{attribute 'hide_all_locals'}
FUNCTION_BLOCK FB_3_COMM_AXIS_BECKHOFF EXTENDS FB_1_COMM
VAR_INPUT
  StopVelocityTolerance : LREAL := 0.000001;
END_VAR
VAR_IN_OUT
    Axis : AXIS_REF;
END_VAR
VAR_OUTPUT
  Powered : BOOL;
  Homed : BOOL;
  ActualPosition : LREAL;
  ActualVelocity : LREAL;
END_VAR
VAR
    _fbPower : MC_Power;
    _fbMoveAbsolute : MC_MoveAbsolute;
    _fbMoveRelative : MC_MoveRelative;
    _fbHome : MC_Home;
    _fbStop : MC_Stop;
    _fbReset : MC_Reset;

    _powerRequest : BOOL;
    _moveAbsExecute : BOOL;
    _moveRelExecute : BOOL;
    _homeExecute : BOOL;
    _stopExecute : BOOL;
    _resetExecute : BOOL;
    _commandAccepted : BOOL;
END_VAR

// ------ CALL CYCLIC -----------------
CYCLIC_COMM();



// ------ WRITE HMI -------------------
		// NO HMI STRUCT

// ------ READ FROM HMI ---------------
		// NO HMI STRUCT
	


// ------ WRITE PROPS/METHODS ---------
Connected := RequestConnection;
Operational := RequestConnection;

CanAcceptCommand := NOT _fbStop.Busy AND NOT _stopExecute AND NOT _resetExecute;


// ----- CALL POUS AND ERROR SURVEILLANCE ----------

_fbPower(Axis := Axis, Enable := _powerRequest, Enable_Positive := _powerRequest, Enable_Negative := _powerRequest);
_fbMoveAbsolute(Axis := Axis, Execute := _moveAbsExecute);
_fbMoveRelative(Axis := Axis, Execute := _moveRelExecute);
_fbHome(Axis := Axis, Execute := _homeExecute);
_fbStop(Axis := Axis, Execute := _stopExecute);
_fbReset(Axis := Axis, Execute := _resetExecute);



IF _fbPower.Error THEN Messenger.AddError(eMessageCategories.HardwareFailure, CONCAT(Path, '.Power'), 'MC_Power error'); END_IF
IF _fbMoveAbsolute.Error THEN Messenger.AddError(eMessageCategories.HardwareFailure, CONCAT(Path, '.MoveAbsolute'), 'MC_MoveAbsolute error'); END_IF
IF _fbMoveRelative.Error THEN Messenger.AddError(eMessageCategories.HardwareFailure, CONCAT(Path, '.MoveRelative'), 'MC_MoveRelative error'); END_IF
IF _fbHome.Error THEN Messenger.AddError(eMessageCategories.HardwareFailure, CONCAT(Path, '.Home'), 'MC_Home error'); END_IF
IF _fbStop.Error THEN Messenger.AddError(eMessageCategories.HardwareFailure, CONCAT(Path, '.Stop'), 'MC_Stop error'); END_IF
IF _fbReset.Error THEN Messenger.AddError(eMessageCategories.HardwareFailure, CONCAT(Path, '.Reset'), 'MC_Reset error'); END_IF


// ----- REST --------------------

Powered := _fbPower.Status;
ActualPosition := Axis.NcToPlc.ActPos;
ActualVelocity := Axis.NcToPlc.ActVelo;


IF Busy AND NOT StopPending THEN
  IF Messenger.HasActivError OR NOT Operational THEN
        _moveAbsExecute := FALSE;
        _moveRelExecute := FALSE;
        _homeExecute := FALSE;
        ActiveCommandID := 0;
        CommandState := eProgress.FINALIZED;
        CommandResult :=eResult.ERROR;
        Busy := FALSE;

    ELSIF _fbMoveAbsolute.CommandAborted OR _fbMoveRelative.CommandAborted OR _fbHome.CommandAborted THEN
        _moveAbsExecute := FALSE;
        _moveRelExecute := FALSE;
        _homeExecute := FALSE;
        ActiveCommandID := 0;
        CommandState := eProgress.ABORTED;
        CommandResult :=eResult.FAILURE;
        Busy := FALSE;

    ELSIF _fbMoveAbsolute.Done OR _fbMoveRelative.Done OR _fbHome.Done THEN
        IF _fbHome.Done THEN Homed := TRUE; END_IF
        _moveAbsExecute := FALSE;
        _moveRelExecute := FALSE;
        _homeExecute := FALSE;
        ActiveCommandID := 0;
        CommandState := eProgress.FINALIZED;
        CommandResult :=eResult.SUCCESS;
        Busy := FALSE;

    ELSIF NOT _commandAccepted AND (_fbMoveAbsolute.Busy OR _fbMoveRelative.Busy OR _fbHome.Busy) THEN
        _commandAccepted := TRUE;
        AcceptedCommandID := ActiveCommandID;
        CommandState := eProgress.ACKNOWLEDGE;
        _moveAbsExecute := FALSE;
        _moveRelExecute := FALSE;
        _homeExecute := FALSE;
    ELSIF _commandAccepted AND (_fbMoveAbsolute.Busy OR _fbMoveRelative.Busy OR _fbHome.Busy) THEN
        CommandState := eProgress.RUNNING;
    END_IF
END_IF

IF _fbStop.Done OR _fbStop.CommandAborted OR _fbStop.Error THEN _stopExecute := FALSE; END_IF
IF _fbReset.Done OR _fbReset.Error THEN _resetExecute := FALSE; END_IF

METHOD PROTECTED HasPhysicalStopFailed : BOOL
HasPhysicalStopFailed := _fbStop.Error OR _fbStop.CommandAborted;
END_METHOD

METHOD PROTECTED IsPhysicalStopComplete : BOOL
IsPhysicalStopComplete :=
    _fbStop.Done
    AND (ABS(ActualVelocity) <= StopVelocityTolerance);
END_METHOD

PROPERTY Operational : BOOL
SET
SUPER^.Operational := Operational;
END_SET
END_PROPERTY

METHOD PUBLIC Power : BOOL
VAR_INPUT Enable : BOOL; END_VAR
_powerRequest := Enable;
Power := TRUE;
END_METHOD

METHOD PUBLIC ResetAxis : BOOL
_resetExecute := TRUE;
ResetAxis := TRUE;
END_METHOD

METHOD PUBLIC ResetCommunication : BOOL
_moveAbsExecute := FALSE;
_moveRelExecute := FALSE;
_homeExecute := FALSE;
_stopExecute := FALSE;
AcceptedCommandID := 0;
ActiveCommandID := 0;

CommandState := eProgress.INIT;
CommandResult :=eResult.NONE;
Reconnect();
ResetCommunication := TRUE;
END_METHOD

METHOD PUBLIC SendHome : BOOL
VAR_INPUT CommandID : UINT; END_VAR
SendHome := FALSE;
IF (CommandID = 0) OR NOT CanAcceptCommand THEN RETURN; END_IF
Homed := FALSE;
_homeExecute := TRUE;
_commandAccepted := FALSE;
AcceptedCommandID := 0;
ActiveCommandID := CommandID;
CommandState := eProgress.INIT;
CommandResult :=eResult.NONE;
SendHome := TRUE;
END_METHOD

METHOD PUBLIC SendMoveAbsolute : BOOL
VAR_INPUT
    CommandID : UINT; Position : LREAL; Velocity : LREAL; Acceleration : LREAL; Deceleration : LREAL; Jerk : LREAL;
END_VAR
SendMoveAbsolute := FALSE;
IF (CommandID = 0) OR NOT CanAcceptCommand THEN RETURN; END_IF
_fbMoveAbsolute.Position := Position;
_fbMoveAbsolute.Velocity := Velocity;
_fbMoveAbsolute.Acceleration := Acceleration;
_fbMoveAbsolute.Deceleration := Deceleration;
_fbMoveAbsolute.Jerk := Jerk;
_moveAbsExecute := TRUE;
_commandAccepted := FALSE;
AcceptedCommandID := 0;
ActiveCommandID := CommandID;
CommandState := eProgress.INIT;
CommandResult :=eResult.NONE;
SendMoveAbsolute := TRUE;
END_METHOD

METHOD PUBLIC SendMoveRelative : BOOL
VAR_INPUT
    CommandID : UINT; Distance : LREAL; Velocity : LREAL; Acceleration : LREAL; Deceleration : LREAL; Jerk : LREAL;
END_VAR
SendMoveRelative := FALSE;
IF (CommandID = 0) OR NOT CanAcceptCommand THEN RETURN; END_IF
_fbMoveRelative.Distance := Distance;
_fbMoveRelative.Velocity := Velocity;
_fbMoveRelative.Acceleration := Acceleration;
_fbMoveRelative.Deceleration := Deceleration;
_fbMoveRelative.Jerk := Jerk;
_moveRelExecute := TRUE;
_commandAccepted := FALSE;
AcceptedCommandID := 0;
ActiveCommandID := CommandID;
CommandState := eProgress.INIT;
CommandResult :=eResult.NONE;
SendMoveRelative := TRUE;
END_METHOD

METHOD PROTECTED StartPhysicalStop : BOOL
VAR_INPUT
    Mode : eStopMode;
END_VAR
StartPhysicalStop := FALSE;
IF NOT Connected THEN
    RETURN;
END_IF

_moveAbsExecute := FALSE;
_moveRelExecute := FALSE;
_homeExecute := FALSE;
_stopExecute := TRUE;
StartPhysicalStop := TRUE;
END_METHOD

METHOD PUBLIC StopMotion : BOOL
StopMotion := SUPER^.StopMotion();
END_METHOD

END_FUNCTION_BLOCK

(* stored: Version 1.1.0.1, ProductVersion 3.1.4026.18
   POU FB_3_COMM_AXIS_BECKHOFF: Id {6590ca91-e828-49ed-96d5-a1b6fe08b87c}, SpecialFunc None
   Method HasPhysicalStopFailed: Id {07ba1865-cb6a-4a8c-96a0-eef840195aa0}
   Method IsPhysicalStopComplete: Id {a22113a2-02df-430f-b71d-3b7827035089}
   Property Operational: Id {4e3d4c82-6c3e-4a6a-814a-07ce7bf49eff}
   Set Set: Id {a12a9d16-3a48-4fe1-b1c6-4b5bb26f80c2}
   Method Power: Id {5009c6e1-2c2e-4e9f-8bd0-48ea7245eeb8}
   Method ResetAxis: Id {8993a558-2273-4b75-9edd-81b579dc1f02}
   Method ResetCommunication: Id {d6df4f8c-4fb8-47c4-8972-2548e217db7f}
   Method SendHome: Id {bc5b9968-2431-457c-aab0-516da2c5d033}
   Method SendMoveAbsolute: Id {5b81aea5-0ab7-4117-8b92-2d5fae6e40c0}
   Method SendMoveRelative: Id {8db40419-b654-4ba0-9a9d-02d59aa67ced}
   Method StartPhysicalStop: Id {a2ac5ac5-15e0-4ed8-95b0-80d6f3ff3736}
   Method StopMotion: Id {c0fae11f-2aa8-4051-9726-2a746e1e0326} *)
